INTERFACE PUBLIC ExecuteCommands EXTENDS RunningStateCommands, ActionStateCommands, HoldableStateCommands

METHOD PUBLIC Suspend
END_METHOD

END_INTERFACE

(* stored: Version 1.1.0.1, ProductVersion 3.1.4026.18
   Itf ExecuteCommands: Id {9dab06e0-c06a-0aec-34db-a51978aa62c9}
   Method Suspend: Id {2f703afa-fea1-0aae-04b9-1ccf0ad65f2e} *)
